{attribute 'TcGenerated'}
{attribute 'no-analysis'}
{attribute 'linkalways'}
// This function has been automatically generated from the project information.
VAR_GLOBAL CONSTANT
	{attribute 'const_non_replaced'}
	stLibVersion_Strings : ST_LibVersion := (iMajor := 0, iMinor := 0, iBuild := 1, iRevision := 0, nFlags := 0, sVersion := '0.0.1');
END_VAR

(* stored: Version 1.1.0.1, ProductVersion 3.1.4024.12
   GVL Global_Version: Id {d824f2c3-2a50-417d-8da2-7f0496cb2c16} *)
